(* PLC project Tc2_Utilities.FB_GetHostName Demo, tc3-libraries-kb TwinCAT 3.1 *)
(* stored: creationDateTime 2026-05-11T00:00:00, modificationDateTime 2026-05-11T00:00:00 *)

PROGRAM P_Demo_FB_GetHostName
  VAR
    fbFB_GetHostName : FB_GetHostName;  (* FB_GetHostName 实例 *)
    bRead : BOOL := FALSE;
    sName : STRING;
    bBusy_ : BOOL;
    bErrFlag : BOOL;
    nErrCode : UDINT;
  END_VAR

// =============================================================================
// 场景：开机后读机器名给 HMI 标题。
// 价值：标准库调用，免写注册表读取。
// 验证：改 bRead := TRUE，观察 sName 装载主机名字符串。
// 验证步骤：
//   1. 右键 PLC 项目 → Import PLCopenXML → 选本文件
//   2. 引用 Tc2_Utilities（References → Add library）
//   3. 编译 → 登录 → 运行；按上方『验证』行的指示在线写值观察
// =============================================================================

fbFB_GetHostName(
    bExecute := bRead,
    tTimeout := DEFAULT_ADS_TIMEOUT,
    sHostName => sName,
    bBusy => bBusy_,
    bErr => bErrFlag,
    nErrId => nErrCode
);
END_PROGRAM
